# EPICS autosave request: as/req/modules_I404.req
#FILE... modules_I404.req

file "I404.req", Sys=XF:28IDA-BI:1, Dev={BPM:2}
